# EPICS substitutions: OPCUA/OPCUA-IOC-01App/Db/Merlin_vacuum.substitutions
global{NS="\$(NS)",P="\$(P)",SUBS="\$(SUBS)",DEBUG="\$(DEBUG=0)"}
file "$(TOP)/OPCUA-IOC-01App/Db/MAPS_vacuum.template" {
	pattern{ RECORD_TYPE, PV_NAME, NAME_PREFIX, NAME_SUFFIX}
	{ "stringin", "PE_UNDERRANGE", "\$(NAME_PREFIX)", "Statuses.PE_Underrange_Control" }
    { "stringin", "UNIT", "\$(NAME_PREFIX)", "Statuses.Pressure_Unit" }
    { "stringin", "ERROR", "\$(NAME_PREFIX)", "Statuses.TPG_Error" }
    { "bi", "HEALTHY", "\$(NAME_PREFIX)", "Statuses.TPG_Healthy" }
	{ "bi", "COMMS_ERROR", "\$(NAME_PREFIX)", "Statuses.Comms_Error" }

    { "ai", "PRESSURE_A1", "\$(NAME_PREFIX)", "Sensor_A1.Pressure" }
    { "stringin", "MEASURED_VALUE_A1", "\$(NAME_PREFIX)", "Sensor_A1.Measured_Value_Status" }
    { "stringin", "MEASURING_CIRCUIT_A1", "\$(NAME_PREFIX)", "Sensor_A1.Measuring_Circuit_Status" }
    { "stringin", "FILTER_TIME_CONST_A1", "\$(NAME_PREFIX)", "Sensor_A1.Filter_Time_Constant" }
	{ "stringin", "NAME_A1", "\$(NAME_PREFIX)", "Sensor_A1.Name" }
	{ "ai", "THRESHOLD_LOW_A1", "\$(NAME_PREFIX)", "Relay1.Lower_Threshold" }
    { "ai", "THRESHOLD_HI_A1", "\$(NAME_PREFIX)", "Relay1.Upper_Threshold" }
	{ "stringin", "SWITCH_FUNC_ASSIGN_A1", "\$(NAME_PREFIX)", "Relay1.Switching_Function_Assignment" }
    { "stringin", "SWITCH_FUNC_STATUS_A1", "\$(NAME_PREFIX)", "Relay1.Switching_Function_Status" }

    { "ai", "PRESSURE_A2", "\$(NAME_PREFIX)", "Sensor_A2.Pressure" }
	{ "stringin", "MEASURED_VALUE_A2", "\$(NAME_PREFIX)", "Sensor_A2.Measured_Value_Status" }
    { "stringin", "MEASURING_CIRCUIT_A2", "\$(NAME_PREFIX)", "Sensor_A2.Measuring_Circuit_Status" }
	{ "stringin", "FILTER_TIME_CONST_A2", "\$(NAME_PREFIX)", "Sensor_A2.Filter_Time_Constant" }
	{ "stringin", "NAME_A2", "\$(NAME_PREFIX)", "Sensor_A2.Name" }
    { "ai", "THRESHOLD_LOW_A2", "\$(NAME_PREFIX)", "Relay2.Lower_Threshold" }
    { "ai", "THRESHOLD_HI_A2", "\$(NAME_PREFIX)", "Relay2.Upper_Threshold" }
    { "stringin", "SWITCH_FUNC_ASSIGN_A2", "\$(NAME_PREFIX)", "Relay2.Switching_Function_Assignment" }
    { "stringin", "SWITCH_FUNC_STATUS_A2", "\$(NAME_PREFIX)", "Relay2.Switching_Function_Status" }

    { "ai", "PRESSURE_B1", "\$(NAME_PREFIX)", "Sensor_B1.Pressure" }
    { "stringin", "MEASURED_VALUE_B1", "\$(NAME_PREFIX)", "Sensor_B1.Measured_Value_Status" }
    { "stringin", "MEASURING_CIRCUIT_B1", "\$(NAME_PREFIX)", "Sensor_B1.Measuring_Circuit_Status" }
    { "stringin", "FILTER_TIME_CONST_B1", "\$(NAME_PREFIX)", "Sensor_B1.Filter_Time_Constant" }
	{ "stringin", "NAME_B1", "\$(NAME_PREFIX)", "Sensor_B1.Name" }
    { "ai", "THRESHOLD_LOW_B1", "\$(NAME_PREFIX)", "Relay3.Lower_Threshold" }
    { "ai", "THRESHOLD_HI_B1", "\$(NAME_PREFIX)", "Relay3.Upper_Threshold" }
    { "stringin", "SWITCH_FUNC_ASSIGN_B1", "\$(NAME_PREFIX)", "Relay3.Switching_Function_Assignment" }
    { "stringin", "SWITCH_FUNC_STATUS_B1", "\$(NAME_PREFIX)", "Relay3.Switching_Function_Status" }

    { "ai", "PRESSURE_B2", "\$(NAME_PREFIX)", "Sensor_B2.Pressure" }
    { "stringin", "MEASURED_VALUE_B2", "\$(NAME_PREFIX)", "Sensor_B2.Measured_Value_Status" }
    { "stringin", "MEASURING_CIRCUIT_B2", "\$(NAME_PREFIX)", "Sensor_B2.Measuring_Circuit_Status" }
    { "stringin", "FILTER_TIME_CONST_B2", "\$(NAME_PREFIX)", "Sensor_B2.Filter_Time_Constant" }
	{ "stringin", "NAME_B2", "\$(NAME_PREFIX)", "Sensor_B2.Name" }
    { "ai", "THRESHOLD_LOW_B2", "\$(NAME_PREFIX)", "Relay4.Lower_Threshold" }
    { "ai", "THRESHOLD_HI_B2", "\$(NAME_PREFIX)", "Relay4.Upper_Threshold" }
    { "stringin", "SWITCH_FUNC_ASSIGN_B2", "\$(NAME_PREFIX)", "Relay4.Switching_Function_Assignment" }
    { "stringin", "SWITCH_FUNC_STATUS_B2", "\$(NAME_PREFIX)", "Relay4.Switching_Function_Status" }

}
